Staubli VAL3: MotionQueue.pjx

--- MotionQueue.pjx ---
Parameters version=s7.7.2 stackSize=5000 millimeterUnit=true
Program file=getNumElements.pgx
Program file=pop.pgx
Program file=push.pgx
Program file=push_front.pgx
Program file=start.pgx
Program file=stop.pgx
Data file=MotionQueue.dtx
Type name=MotionBuffer path=Disk://MotionBuffer/MotionBuffer.pjx

--- MotionQueue.dtx ---
public num nPush
public num nPop
public num nElems
public MotionBuffer buffer[10]
  [0]
    mdesc mVelAcc = {leave=0, reach=0}
    num nDuration
    num nSequence
    jointRx jJointRx
  [1]
    mdesc mVelAcc = {leave=0, reach=0}
    num nDuration
    num nSequence
    jointRx jJointRx
  [2]
    mdesc mVelAcc = {leave=0, reach=0}
    num nDuration
    num nSequence
    jointRx jJointRx
  [3]
    mdesc mVelAcc = {leave=0, reach=0}
    num nDuration
    num nSequence
    jointRx jJointRx
  [4]
    mdesc mVelAcc = {leave=0, reach=0}
    num nDuration
    num nSequence
    jointRx jJointRx
  [5]
    mdesc mVelAcc = {leave=0, reach=0}
    num nDuration
    num nSequence
    jointRx jJointRx
  [6]
    mdesc mVelAcc = {leave=0, reach=0}
    num nDuration
    num nSequence
    jointRx jJointRx
  [7]
    mdesc mVelAcc = {leave=0, reach=0}
    num nDuration
    num nSequence
    jointRx jJointRx
  [8]
    mdesc mVelAcc = {leave=0, reach=0}
    num nDuration
    num nSequence
    jointRx jJointRx
  [9]
    mdesc mVelAcc = {leave=0, reach=0}
    num nDuration
    num nSequence
    jointRx jJointRx

--- start.pgx ---
program start()
begin
  nPush = 0
  nPop = 0
  nElems = 0
end

--- clear.pgx ---
public program clear()
begin
  nElems = 0
  nPush = nPop
end

--- push.pgx ---
public program push(MotionBuffer& x_cmd, bool& x_res)
begin
  if (nElems < size(buffer))
    buffer[nPush] = x_cmd
    nElems = nElems + 1
    nPush = nPush + 1
    if (nPush >= size(buffer))
      nPush = 0
    endIf
    x_res = true
  else
    x_res = false
  endIf
end

--- push_front.pgx ---
public program push_front(bool& x_res, MotionBuffer& x_cmd)
begin
end
